FUNCTION_BLOCK NeredaSludgeBuffer_2 (* Composite Function Block Type *)
  (* Standard: 61499-2 *)
  (* Version 1.1, 9/30/2026, Claude/Hidryco, Schneider Electric, Rev1.1 - Religadas as 4 conexoes do 49FT0004 (PV2..PV5 -> FlowMeasurement_SD1/SD2/WD1/WD2) *)
  PACKAGE SE.Nereda;
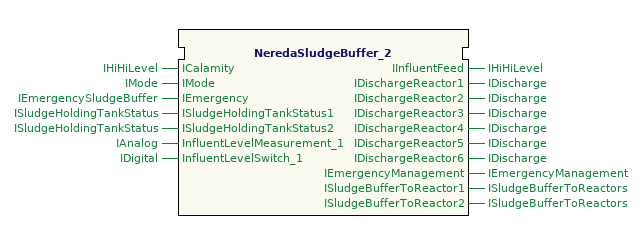
  SOCKETS
    ICalamity : IHiHiLevel;
    IMode : IMode;
    IEmergency : IEmergencySludgeBuffer;
    ISludgeHoldingTankStatus1 : ISludgeHoldingTankStatus;
    ISludgeHoldingTankStatus2 : ISludgeHoldingTankStatus;
    InfluentLevelMeasurement_1 : IAnalog;
    InfluentLevelSwitch_1 : IDigital;
  END_SOCKETS
  PLUGS
    IInfluentFeed : IHiHiLevel;
    IDischargeReactor1 : IDischarge;
    IDischargeReactor2 : IDischarge;
    IDischargeReactor3 : IDischarge;
    IDischargeReactor4 : IDischarge;
    IDischargeReactor5 : IDischarge;
    IDischargeReactor6 : IDischarge;
    IEmergencyManagement : IEmergencyManagement;
    ISludgeBufferToReactor1 : ISludgeBufferToReactors;
    ISludgeBufferToReactor2 : ISludgeBufferToReactors;
  END_PLUGS
  (* 01 - FUNCTIONNAL INPUT INTERFACE *)
  (* 00 - INITIALIZATION *)
  (* 05 - LOGIC *)
  (* 06 - HMI INTERFACE *)
  (* 03 - FIELD INTERFACE *)
  (* 02 - FUNCTIONNAL OUTPUT INTERFACE *)
  (* Sludge Buffer Logic *)
  (* 04 - CHILDREN *)
  (* 4A - TYPICALS *)
  FBS
    IThis : NeredaSludgeBuffer_2_HMI(QI := TRUE);
    INIT : plcStart(Prio := 50, Delay := T#0ms);
    Logic : SludgeBufferLogic_2; {SET_ATTRIBUTE(Configuration.Component.HideUnusedPorts, )}
    Actuators : SludgeBufferActuators_2;
    Sensors : SludgeBufferSensors_2;
  END_FBS
  EVENT_CONNECTIONS
    Actuators.INITO TO Logic.INIT;
    Logic.INITO TO INIT.ACK_FIRST;
    Sensors.INITO TO Actuators.INIT;
    INIT.FIRST_INIT TO IThis.375FA441A12CD8F1;
    INIT.REDO_INIT TO IThis.375FA441A12CD8F1;
    Sensors.8A212303AC297946 TO IThis.F15236EC377513F4;
    IThis.BBCA781EE0906F6D TO Sensors.INIT;
  END_CONNECTIONS
  DATA_CONNECTIONS
    Sensors.C5C1B8B409063B7A TO IThis.04E0874FDDD12A13;
    Sensors.6DED050C37342A8D TO IThis.DF0AD27AB0A501A4;
  END_CONNECTIONS
  ADAPTER_CONNECTIONS
    ICalamity TO Logic.57C6A46265899F0E;
    Logic.E34663B92C032BE3 TO IInfluentFeed;
    Logic.65CD2892A8390CC7 TO IDischargeReactor1;
    Logic.09733019B81C471D TO IDischargeReactor2;
    Logic.9BA7D7F1ED9A24F4 TO Actuators.D5C49F7D36A7EF36;
    Logic.AAC7A3CC2063C695 TO Actuators.CC8D4552F6D34008;
    Logic.C630E5646368B2F6 TO Actuators.A1591D94EED364EB;
    Logic.CC2C61EF84F8343D TO Actuators.84E92E0AC3FBE059;
    Logic.49614280FF6DD736 TO Actuators.448CD69762F3560D;
    Logic.B75D31F2B8B725A7 TO Actuators.0D1F85112FC02318;
    Logic.557F5BA18E16352C TO Actuators.CE1734A2D1856938;
    Logic.DB6554290D3E07B3 TO Actuators.64631004EDA33B2B;
    Logic.6101DA11469C8453 TO Actuators.BED0F4622A613B55;
    Logic.004A012418AA2C01 TO Actuators.31A0A14FC5769DD7;
    Logic.085EF5E3057740C2 TO Actuators.A4ACF8BE4CDA9557;
    Logic.7003DBCF68D589A0 TO Actuators.9550F75AF67D63CC;
    Sensors.DB371618570B635A TO Logic.B6B2ED85FF741ABC;
    Sensors.FC3C623EDF286130 TO Logic.DB9C55C4729EC0EA;
    Sensors.FCC7DD23D033A27A TO Logic.5703C23C77CCE961;
    Sensors.614559B1CCCFFDF4 TO Logic.EFEDE598BC2FC200;
    Logic.3DA9624087A74DA7 TO Actuators.381770F6513B7A86;
    Logic.212CF4265877622F TO Actuators.53EF1DB30A62913C;
    Logic.D68F960858A2E969 TO IDischargeReactor3;
    Logic.B03CF563FA94B299 TO IDischargeReactor4;
    Logic.EC9597B1339EDAF5 TO IDischargeReactor5;
    Logic.3270CCD359089F5D TO IDischargeReactor6;
    Actuators.84480A95EAFBB743 TO Logic.F49C543F5C002B3D;
    Actuators.FB27FBA917E247EA TO Logic.0F671A8319403079;
    Actuators.A32BBA75A2AB451A TO Logic.F62F6370ED41F2AF;
    Actuators.097BE6165BCBF4F4 TO Logic.D800C00007211F89;
    Actuators.73A274DB9C0CA91C TO Logic.B7FDD6B2DD6DEA25;
    Actuators.4516253B740B0B9D TO Logic.646022188B7A14BE;
    Actuators.6C495B9B2BFC34AD TO Logic.075D3971D246343C;
    Actuators.B45B37B0049325DD TO Logic.5363AC234407766A;
    Actuators.9225142A239F7C54 TO Logic.CB9B02A84129EBB6;
    Actuators.B184DEE2B4C16E7D TO Logic.20ACC80485DAEEAE;
    Logic.BC0BF25EE2B28DE8 TO Actuators.C6C634B8D0FF3554;
    Logic.B196818A14AFC35F TO Actuators.0833834A82682CD5;
    Logic.882BF6BCB320A6AD TO Actuators.3520F74F052789BA;
    IMode TO Logic.5BE5DD81D4B3A63E;
    Logic.DB49A38F5A687571 TO IEmergencyManagement;
    Actuators.19623D1DAB015EC1 TO Logic.F4CF4F0009C9569B;
    Actuators.01D3D02BDA029316 TO Logic.E1BEB14A8F3A2EDA;
    Actuators.26F9642B3AA39834 TO Logic.B6A5D01852FFE7AB;
    Actuators.84BB0BAE633E8457 TO Logic.4ECBB77843F57D24;
    Sensors.4D7B45FFF47C623B TO Logic.63D49B7917D98070;
    Sensors.B6F62DFCDA42B53B TO Logic.0C367882A1D9F11A;
    ISludgeHoldingTankStatus1 TO Logic.F31CD366A9C6B9C0;
    ISludgeHoldingTankStatus2 TO Logic.DEA61418023D2E43;
    InfluentLevelMeasurement_1 TO Logic.CBD3FAE12EAD87A2;
    InfluentLevelSwitch_1 TO Logic.DC5AC7E7DE53295E;
    Logic.D2041060D3E6DC4A TO ISludgeBufferToReactor1;
    Logic.7478B5F565D8EB13 TO ISludgeBufferToReactor2;
    IEmergency TO Logic.60E2A1E0C2F716DD;
    Logic.76E25A840C2754A6 TO Actuators.F0ECB7B76630BC75;
    Actuators.5234AFF3EEE9A7DB TO Logic.E471CC5C802B9550;
    Sensors.9E482EEF2D30CEF0 TO Logic.D3F803F9B98F2886;
    Sensors.40C53B36DDFF2F8B TO Logic.B7756FC109EEC807;
    Sensors.6BBE55CE1ECF37D3 TO Logic.82B7FCF81FB7A138;
    Sensors.D6CAEC20D45C707B TO Logic.7FF9C8335038877A;
  END_CONNECTIONS
END_FUNCTION_BLOCK
